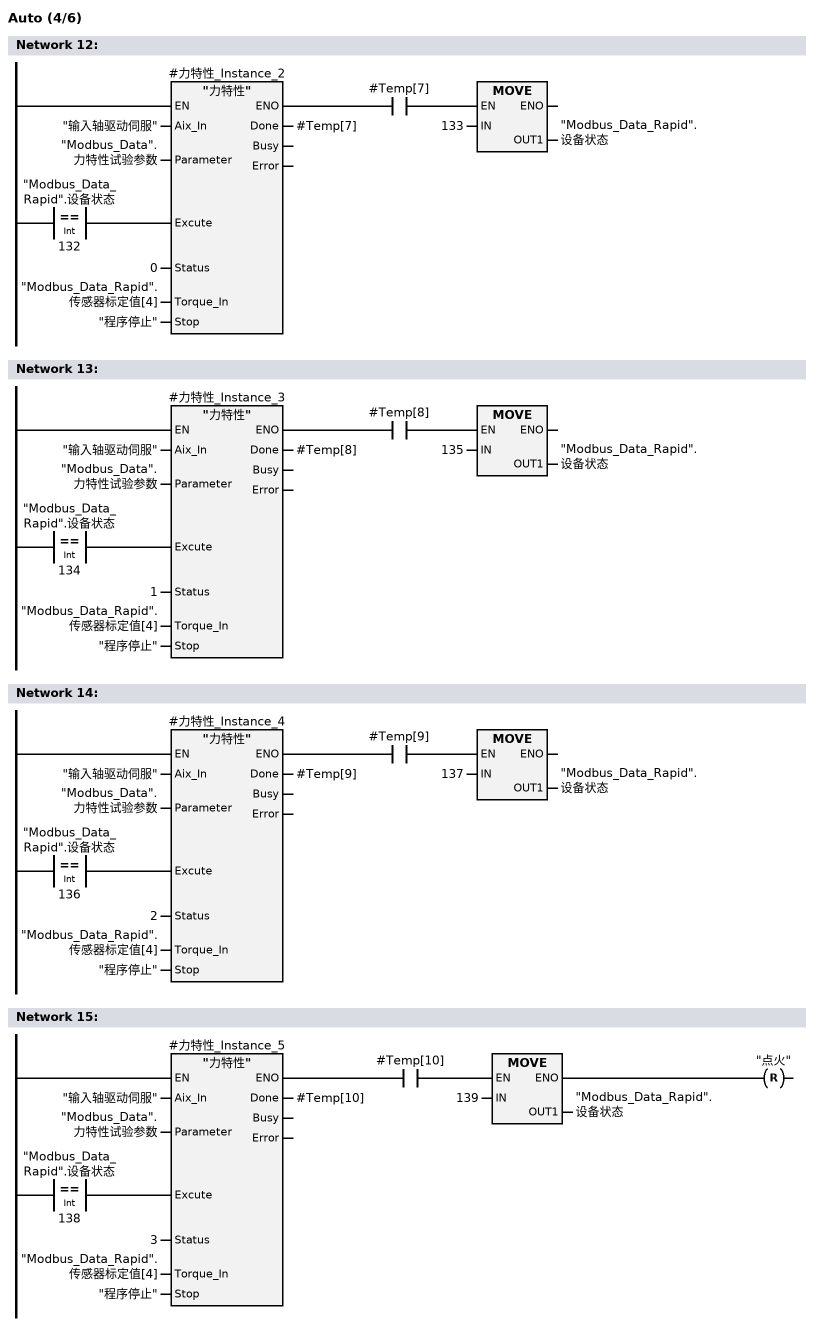
   RUNG wire#powerrail
      #力特性_Instance_2(Excute := wire#w1, Aix_In := "输入轴驱动伺服", Parameter := "Modbus_Data".力特性试验参数, Status := 0, Torque_In := "Modbus_Data_Rapid".传感器标定值[4], Stop := "程序停止", Done => #Temp[7], Busy =>, Error =>)
      Contact( #Temp[7] )
      Move(in := 133, out1 => "Modbus_Data_Rapid".设备状态)
   END_RUNG
   RUNG wire#powerrail
      { S7_Templates := "SrcType := Int" } EQ_Contact(in1 := "Modbus_Data_Rapid".设备状态, in2 := 132)
   END_RUNG wire#w1
   // the same network as SCL:
   #力特性_Instance_2(Aix_In := "输入轴驱动伺服",   // "力特性"
                   Parameter := "Modbus_Data".力特性试验参数,
                   Excute := "Modbus_Data_Rapid".设备状态 = 132,
                   Status := 0,
                   Torque_In := "Modbus_Data_Rapid".传感器标定值[4],
                   Stop := "程序停止",
                   Done => #Temp[7],
                   ENO => #_w1);
   IF #_w1 AND #Temp[7] THEN "Modbus_Data_Rapid".设备状态 := 133; END_IF;
END_REGION

REGION Network 13
   RUNG wire#powerrail
      #力特性_Instance_3(Excute := wire#w1, Aix_In := "输入轴驱动伺服", Parameter := "Modbus_Data".力特性试验参数, Status := 1, Torque_In := "Modbus_Data_Rapid".传感器标定值[4], Stop := "程序停止", Done => #Temp[8], Busy =>, Error =>)
      Contact( #Temp[8] )
      Move(in := 135, out1 => "Modbus_Data_Rapid".设备状态)
   END_RUNG
   RUNG wire#powerrail
      { S7_Templates := "SrcType := Int" } EQ_Contact(in1 := "Modbus_Data_Rapid".设备状态, in2 := 134)
   END_RUNG wire#w1
   // the same network as SCL:
   #力特性_Instance_3(Aix_In := "输入轴驱动伺服",   // "力特性"
                   Parameter := "Modbus_Data".力特性试验参数,
                   Excute := "Modbus_Data_Rapid".设备状态 = 134,
                   Status := 1,
                   Torque_In := "Modbus_Data_Rapid".传感器标定值[4],
                   Stop := "程序停止",
                   Done => #Temp[8],
                   ENO => #_w1);
   IF #_w1 AND #Temp[8] THEN "Modbus_Data_Rapid".设备状态 := 135; END_IF;
END_REGION

REGION Network 14
   RUNG wire#powerrail
      #力特性_Instance_4(Excute := wire#w1, Aix_In := "输入轴驱动伺服", Parameter := "Modbus_Data".力特性试验参数, Status := 2, Torque_In := "Modbus_Data_Rapid".传感器标定值[4], Stop := "程序停止", Done => #Temp[9], Busy =>, Error =>)
      Contact( #Temp[9] )
      Move(in := 137, out1 => "Modbus_Data_Rapid".设备状态)
   END_RUNG
   RUNG wire#powerrail
      { S7_Templates := "SrcType := Int" } EQ_Contact(in1 := "Modbus_Data_Rapid".设备状态, in2 := 136)
   END_RUNG wire#w1
   // the same network as SCL:
   #力特性_Instance_4(Aix_In := "输入轴驱动伺服",   // "力特性"
                   Parameter := "Modbus_Data".力特性试验参数,
                   Excute := "Modbus_Data_Rapid".设备状态 = 136,
                   Status := 2,
                   Torque_In := "Modbus_Data_Rapid".传感器标定值[4],
                   Stop := "程序停止",
                   Done => #Temp[9],
                   ENO => #_w1);
   IF #_w1 AND #Temp[9] THEN "Modbus_Data_Rapid".设备状态 := 137; END_IF;
END_REGION

REGION Network 15
   RUNG wire#powerrail
      #力特性_Instance_5(Excute := wire#w1, Aix_In := "输入轴驱动伺服", Parameter := "Modbus_Data".力特性试验参数, Status := 3, Torque_In := "Modbus_Data_Rapid".传感器标定值[4], Stop := "程序停止", Done => #Temp[10], Busy =>, Error =>)
      Contact( #Temp[10] )
      Move(in := 139, out1 => "Modbus_Data_Rapid".设备状态)
      R_Coil( "点火" )
   END_RUNG
   RUNG wire#powerrail
      { S7_Templates := "SrcType := Int" } EQ_Contact(in1 := "Modbus_Data_Rapid".设备状态, in2 := 138)
   END_RUNG wire#w1
   // the same network as SCL:
   #力特性_Instance_5(Aix_In := "输入轴驱动伺服",   // "力特性"
                   Parameter := "Modbus_Data".力特性试验参数,
                   Excute := "Modbus_Data_Rapid".设备状态 = 138,
                   Status := 3,
                   Torque_In := "Modbus_Data_Rapid".传感器标定值[4],
                   Stop := "程序停止",
                   Done => #Temp[10],
                   ENO => #_w1);
   IF #_w1 AND #Temp[10] THEN
       "Modbus_Data_Rapid".设备状态 := 139;
       "点火" := FALSE;
   END_IF;
END_REGION

REGION Network 16
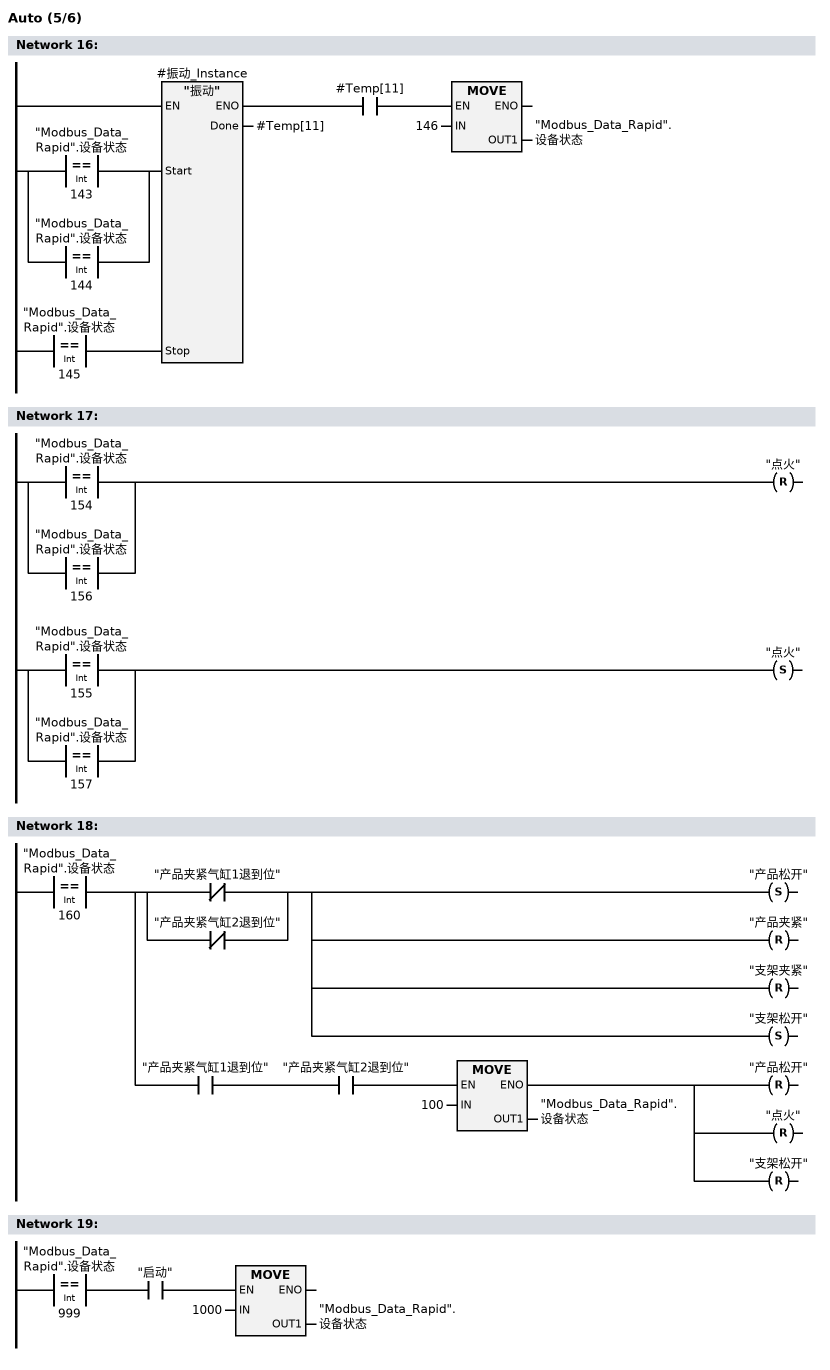
   RUNG wire#powerrail
      #振动_Instance(Start := wire#w1, Stop := wire#w2, Done => #Temp[11])
      Contact( #Temp[11] )
      Move(in := 146, out1 => "Modbus_Data_Rapid".设备状态)
   END_RUNG
   RUNG wire#powerrail
      { S7_Templates := "SrcType := Int" } EQ_Contact(in1 := "Modbus_Data_Rapid".设备状态, in2 := 143)
   END_RUNG wire#w1
   RUNG wire#powerrail
      { S7_Templates := "SrcType := Int" } EQ_Contact(in1 := "Modbus_Data_Rapid".设备状态, in2 := 144)
   END_RUNG wire#w1
   RUNG wire#powerrail
      { S7_Templates := "SrcType := Int" } EQ_Contact(in1 := "Modbus_Data_Rapid".设备状态, in2 := 145)
   END_RUNG wire#w2
   // the same network as SCL:
   #振动_Instance(Start := ("Modbus_Data_Rapid".设备状态 = 143) OR ("Modbus_Data_Rapid".设备状态 = 144),   // "振动"
                Stop := "Modbus_Data_Rapid".设备状态 = 145,
                Done => #Temp[11],
                ENO => #_w1);
   IF #_w1 AND #Temp[11] THEN "Modbus_Data_Rapid".设备状态 := 146; END_IF;
END_REGION

REGION Network 17
   RUNG wire#powerrail
      { S7_Templates := "SrcType := Int" } EQ_Contact(in1 := "Modbus_Data_Rapid".设备状态, in2 := 154)
      wire#w1
      R_Coil( "点火" )
   END_RUNG
   RUNG wire#powerrail
      { S7_Templates := "SrcType := Int" } EQ_Contact(in1 := "Modbus_Data_Rapid".设备状态, in2 := 156)
   END_RUNG wire#w1
   RUNG wire#powerrail
      { S7_Templates := "SrcType := Int" } EQ_Contact(in1 := "Modbus_Data_Rapid".设备状态, in2 := 155)
      wire#w2
      S_Coil( "点火" )
   END_RUNG
   RUNG wire#powerrail
      { S7_Templates := "SrcType := Int" } EQ_Contact(in1 := "Modbus_Data_Rapid".设备状态, in2 := 157)
   END_RUNG wire#w2
   // the same network as SCL:
   IF ("Modbus_Data_Rapid".设备状态 = 154) OR ("Modbus_Data_Rapid".设备状态 = 156) THEN "点火" := FALSE; END_IF;
   IF ("Modbus_Data_Rapid".设备状态 = 155) OR ("Modbus_Data_Rapid".设备状态 = 157) THEN "点火" := TRUE; END_IF;
END_REGION

REGION Network 18
   RUNG wire#powerrail
      { S7_Templates := "SrcType := Int" } EQ_Contact(in1 := "Modbus_Data_Rapid".设备状态, in2 := 160)
      wire#w1
      I_Contact( "产品夹紧气缸1退到位" )
      wire#w2
      S_Coil( "产品松开" )
   END_RUNG
   RUNG wire#w1
      I_Contact( "产品夹紧气缸2退到位" )
   END_RUNG wire#w2
   RUNG wire#w2
      R_Coil( "产品夹紧" )
   END_RUNG
   RUNG wire#w2
      R_Coil( "支架夹紧" )
   END_RUNG
   RUNG wire#w2
      S_Coil( "支架松开" )
   END_RUNG
   RUNG wire#w1
      Contact( "产品夹紧气缸1退到位" )
      Contact( "产品夹紧气缸2退到位" )
      Move(in := 100, out1 => "Modbus_Data_Rapid".设备状态)
      wire#w3
      R_Coil( "产品松开" )
   END_RUNG
   RUNG wire#w3
      R_Coil( "点火" )
   END_RUNG
   RUNG wire#w3
      R_Coil( "支架松开" )
   END_RUNG
   // the same network as SCL:
   #_w1 := "Modbus_Data_Rapid".设备状态 = 160;
   IF #_w1 AND (NOT "产品夹紧气缸1退到位" OR NOT "产品夹紧气缸2退到位") THEN
       "产品松开" := TRUE;
       "产品夹紧" := FALSE;
       "支架夹紧" := FALSE;
       "支架松开" := TRUE;
   END_IF;
   IF #_w1 AND "产品夹紧气缸1退到位" AND "产品夹紧气缸2退到位" THEN
       "Modbus_Data_Rapid".设备状态 := 100;
       "产品松开" := FALSE;
       "点火" := FALSE;
       "支架松开" := FALSE;
   END_IF;
END_REGION

REGION Network 19
   RUNG wire#powerrail
      { S7_Templates := "SrcType := Int" } EQ_Contact(in1 := "Modbus_Data_Rapid".设备状态, in2 := 999)
      Contact( "启动" )
      Move(in := 1000, out1 => "Modbus_Data_Rapid".设备状态)
   END_RUNG
   // the same network as SCL:
   IF ("Modbus_Data_Rapid".设备状态 = 999) AND "启动" THEN "Modbus_Data_Rapid".设备状态 := 1000; END_IF;
END_REGION

REGION Network 20
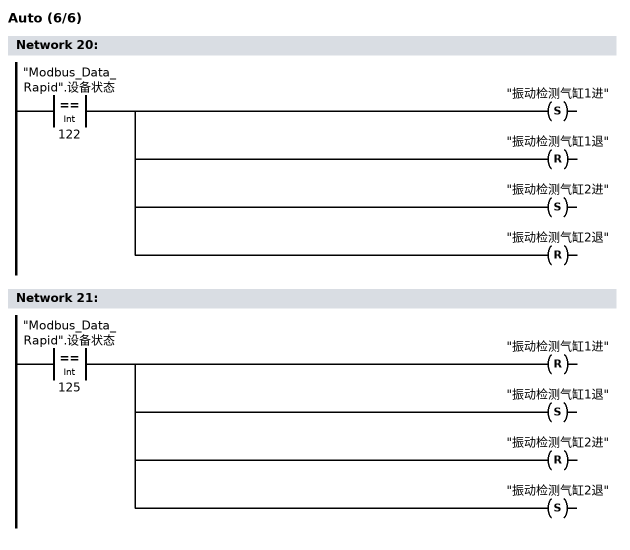
   RUNG wire#powerrail
      { S7_Templates := "SrcType := Int" } EQ_Contact(in1 := "Modbus_Data_Rapid".设备状态, in2 := 122)
      wire#w1
      S_Coil( "振动检测气缸1进" )
   END_RUNG
   RUNG wire#w1
      R_Coil( "振动检测气缸1退" )
   END_RUNG
   RUNG wire#w1
      S_Coil( "振动检测气缸2进" )
   END_RUNG
   RUNG wire#w1
      R_Coil( "振动检测气缸2退" )
   END_RUNG
   // the same network as SCL:
   IF "Modbus_Data_Rapid".设备状态 = 122 THEN
       "振动检测气缸1进" := TRUE;
       "振动检测气缸1退" := FALSE;
       "振动检测气缸2进" := TRUE;
       "振动检测气缸2退" := FALSE;
   END_IF;
END_REGION

REGION Network 21
   RUNG wire#powerrail
      { S7_Templates := "SrcType := Int" } EQ_Contact(in1 := "Modbus_Data_Rapid".设备状态, in2 := 125)
      wire#w1
      R_Coil( "振动检测气缸1进" )
   END_RUNG
   RUNG wire#w1
      S_Coil( "振动检测气缸1退" )
   END_RUNG
   RUNG wire#w1
      R_Coil( "振动检测气缸2进" )
   END_RUNG
   RUNG wire#w1
      S_Coil( "振动检测气缸2退" )
   END_RUNG
   // the same network as SCL:
   IF "Modbus_Data_Rapid".设备状态 = 125 THEN
       "振动检测气缸1进" := FALSE;
       "振动检测气缸1退" := TRUE;
       "振动检测气缸2进" := FALSE;
       "振动检测气缸2退" := TRUE;
   END_IF;
END_REGION
END_FUNCTION_BLOCK

FUNCTION_BLOCK "力特性"   // FB11, LAD
{ S7_Optimized_Access := 'TRUE' }
VERSION : 0.1
   VAR_INPUT
      Aix_In : TO_PositioningAxis;
      Parameter : "Test_Input&Output_Characteristics_CFG";
      Excute : Bool;
      Status : Byte;
      Torque_In : Real;
      Stop : Bool;
   END_VAR
   VAR_OUTPUT
      Done : Bool;
      Busy : Bool;
      Error : Bool;
   END_VAR
   VAR
      "Step" : Int;
      Switch_Torque : Real;
      Test_Velocity : Real;
      Temp : Array[0..7] of Bool;
      MC_Halt_Instance : MC_Halt;
      MC_Home_Instance : MC_Home;
      MC_MoveVelocity_Instance : MC_MoveVelocity;
   END_VAR
   VAR_TEMP   // added for the SCL form of the ladder/FBD networks
      _w1 : Bool;
   END_VAR
BEGIN

REGION Network 1
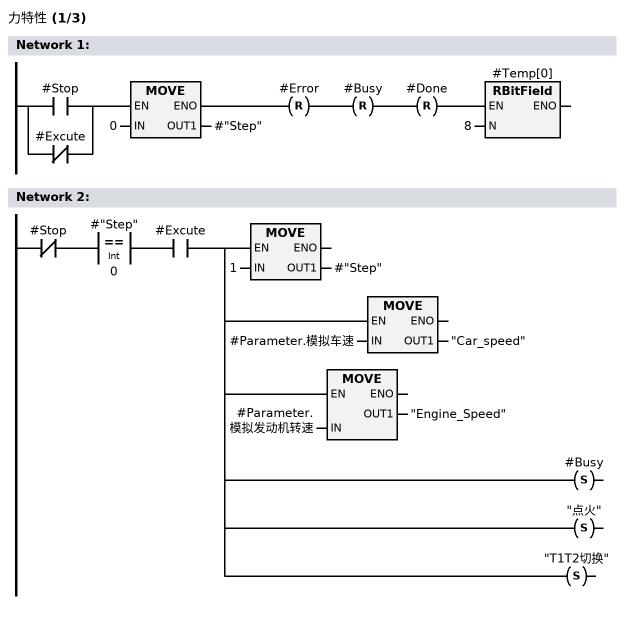
   // no SCL statement known for RBitField: written as a call
   IF #Stop OR NOT #Excute THEN
       #"Step" := 0;
       #Error := FALSE;
       #Busy := FALSE;
       #Done := FALSE;
       RBitField(n := 8, operand := #Temp[0]);
   END_IF;
END_REGION

REGION Network 2
   RUNG wire#powerrail
      I_Contact( #Stop )
      { S7_Templates := "SrcType := Int" } EQ_Contact(in1 := #"Step", in2 := 0)
      Contact( #Excute )
      wire#w1
      Move(in := 1, out1 => #"Step")
   END_RUNG
   RUNG wire#w1
      Move(in := #Parameter.模拟车速, out1 => "Car_speed")
   END_RUNG
   RUNG wire#w1
      Move(in := #Parameter.模拟发动机转速, out1 => "Engine_Speed")
   END_RUNG
   RUNG wire#w1
      S_Coil( #Busy )
   END_RUNG
   RUNG wire#w1
      S_Coil( "点火" )
   END_RUNG
   RUNG wire#w1
      S_Coil( "T1T2切换" )
   END_RUNG
   // the same network as SCL:
   #_w1 := NOT #Stop AND (#"Step" = 0) AND #Excute;
   IF #_w1 THEN
       #"Step" := 1;
       "Car_speed" := #Parameter.模拟车速;
       "Engine_Speed" := #Parameter.模拟发动机转速;
       #Busy := TRUE;
       "点火" := TRUE;
       "T1T2切换" := TRUE;
   END_IF;
END_REGION

REGION Network 3
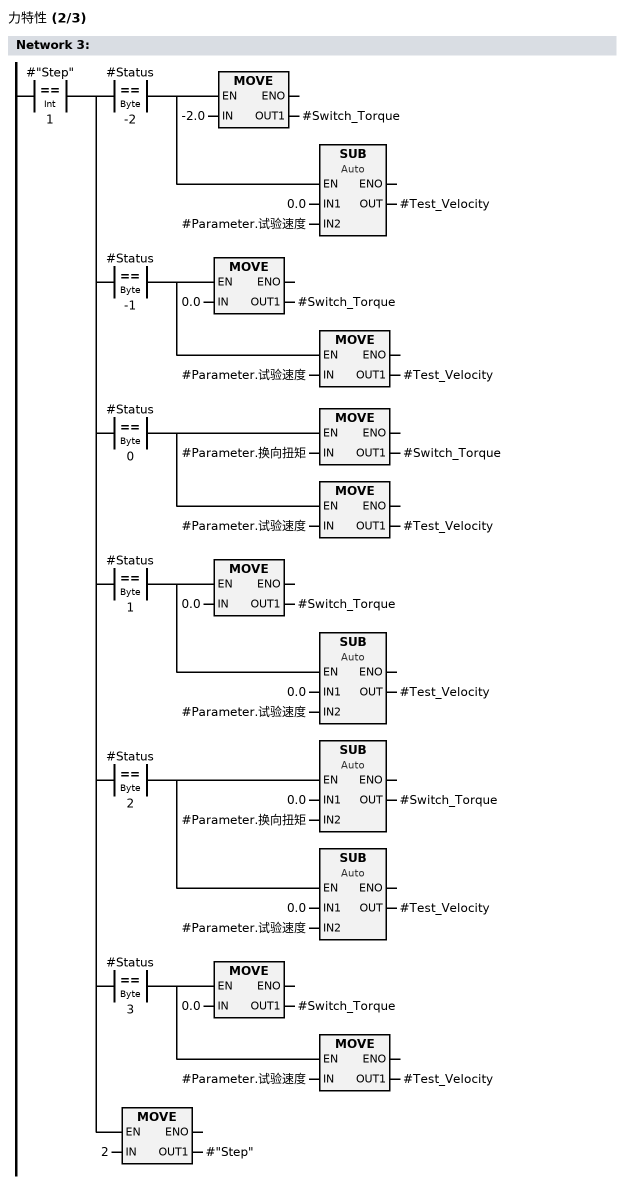
   RUNG wire#powerrail
      { S7_Templates := "SrcType := Int" } EQ_Contact(in1 := #"Step", in2 := 1)
      wire#w1
      { S7_Templates := "SrcType := Byte" } EQ_Contact(in1 := #Status, in2 := -2)
      wire#w2
      Move(in := -2.0, out1 => #Switch_Torque)
   END_RUNG
   RUNG wire#w2
      Sub(in1 := 0.0, in2 := #Parameter.试验速度, out => #Test_Velocity)
   END_RUNG
   RUNG wire#w1
      { S7_Templates := "SrcType := Byte" } EQ_Contact(in1 := #Status, in2 := -1)
      wire#w3
      Move(in := 0.0, out1 => #Switch_Torque)
   END_RUNG
   RUNG wire#w3
      Move(in := #Parameter.试验速度, out1 => #Test_Velocity)
   END_RUNG
   RUNG wire#w1
      { S7_Templates := "SrcType := Byte" } EQ_Contact(in1 := #Status, in2 := 0)
      wire#w4
      Move(in := #Parameter.换向扭矩, out1 => #Switch_Torque)
   END_RUNG
   RUNG wire#w4
      Move(in := #Parameter.试验速度, out1 => #Test_Velocity)
   END_RUNG
   RUNG wire#w1
      { S7_Templates := "SrcType := Byte" } EQ_Contact(in1 := #Status, in2 := 1)
      wire#w5
      Move(in := 0.0, out1 => #Switch_Torque)
   END_RUNG
   RUNG wire#w5
      Sub(in1 := 0.0, in2 := #Parameter.试验速度, out => #Test_Velocity)
   END_RUNG
   RUNG wire#w1
      { S7_Templates := "SrcType := Byte" } EQ_Contact(in1 := #Status, in2 := 2)
      wire#w6
      Sub(in1 := 0.0, in2 := #Parameter.换向扭矩, out => #Switch_Torque)
   END_RUNG
   RUNG wire#w6
      Sub(in1 := 0.0, in2 := #Parameter.试验速度, out => #Test_Velocity)
   END_RUNG
   RUNG wire#w1
      { S7_Templates := "SrcType := Byte" } EQ_Contact(in1 := #Status, in2 := 3)
      wire#w7
      Move(in := 0.0, out1 => #Switch_Torque)
   END_RUNG
   RUNG wire#w7
      Move(in := #Parameter.试验速度, out1 => #Test_Velocity)
   END_RUNG
   RUNG wire#w1
      Move(in := 2, out1 => #"Step")
   END_RUNG
   // the same network as SCL:
   #_w1 := #"Step" = 1;
   IF #_w1 AND (#Status = (-2)) THEN
       #Switch_Torque := -2.0;
       #Test_Velocity := 0.0 - #Parameter.试验速度;
   END_IF;
   IF #_w1 AND (#Status = (-1)) THEN
       #Switch_Torque := 0.0;
       #Test_Velocity := #Parameter.试验速度;
   END_IF;
   IF #_w1 AND (#Status = 0) THEN
       #Switch_Torque := #Parameter.换向扭矩;
       #Test_Velocity := #Parameter.试验速度;
   END_IF;
   IF #_w1 AND (#Status = 1) THEN
       #Switch_Torque := 0.0;
       #Test_Velocity := 0.0 - #Parameter.试验速度;
   END_IF;
   IF #_w1 AND (#Status = 2) THEN
       #Switch_Torque := 0.0 - #Parameter.换向扭矩;
       #Test_Velocity := 0.0 - #Parameter.试验速度;
   END_IF;
   IF #_w1 AND (#Status = 3) THEN
       #Switch_Torque := 0.0;
       #Test_Velocity := #Parameter.试验速度;
   END_IF;
   IF #_w1 THEN #"Step" := 2; END_IF;
END_REGION

REGION Network 4
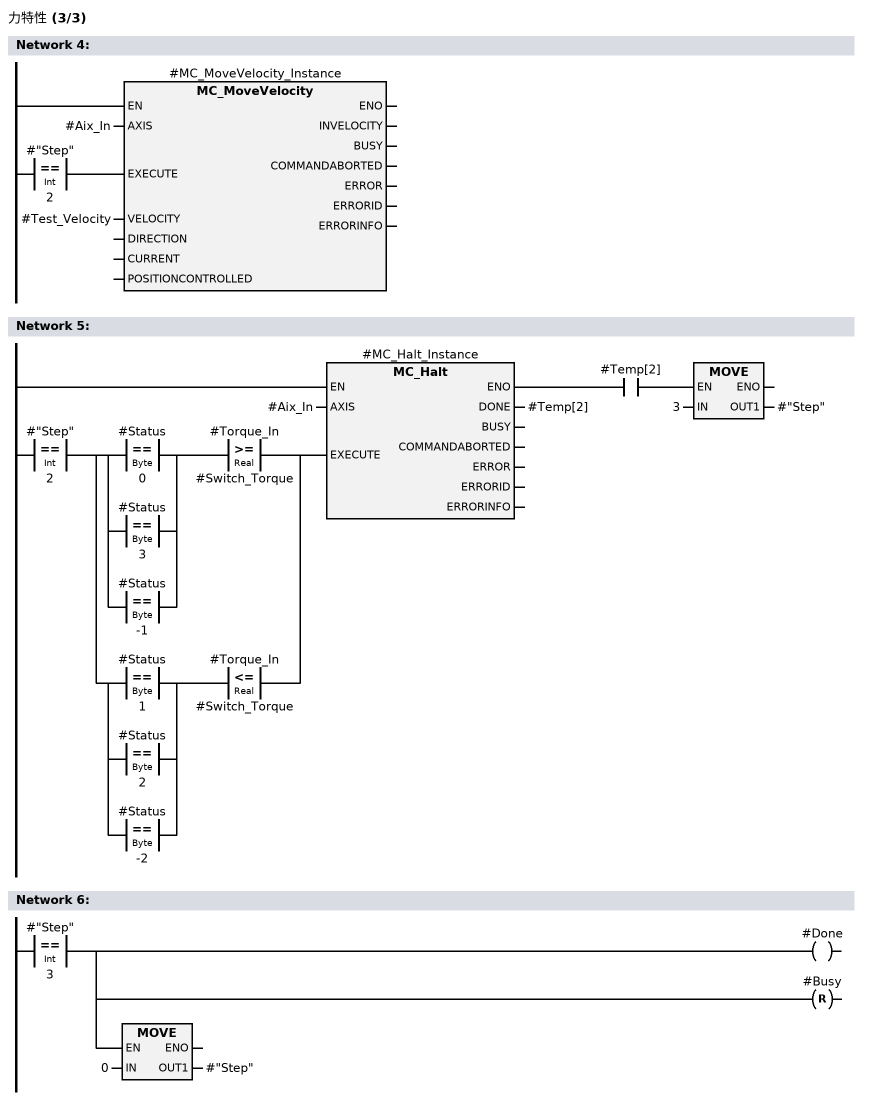
   #MC_MoveVelocity_Instance(Axis := #Aix_In, Execute := #"Step" = 2, Velocity := #Test_Velocity);   // MC_MoveVelocity
END_REGION

REGION Network 5
   // ENO of a box is taken as its EN; it also drops when the box reports an error
   #MC_Halt_Instance(Axis := #Aix_In,   // MC_Halt
                     Execute := (#"Step" = 2) AND ((((#Status = 0) OR (#Status = 3) OR (#Status = (-1))) AND (#Torque_In >= #Switch_Torque)) OR (((#Status = 1) OR (#Status = 2) OR (#Status = (-2))) AND (#Torque_In <= #Switch_Torque))),
                     Done => #Temp[2]);
   IF #Temp[2] THEN #"Step" := 3; END_IF;
END_REGION

REGION Network 6
   RUNG wire#powerrail
      { S7_Templates := "SrcType := Int" } EQ_Contact(in1 := #"Step", in2 := 3)
      wire#w1
      Coil( #Done )
   END_RUNG
   RUNG wire#w1
      R_Coil( #Busy )
   END_RUNG
   RUNG wire#w1
      Move(in := 0, out1 => #"Step")
   END_RUNG
   // the same network as SCL:
   #Done := #"Step" = 3;
   IF #Done THEN
       #Busy := FALSE;
       #"Step" := 0;
   END_IF;
END_REGION
END_FUNCTION_BLOCK

FUNCTION_BLOCK "振动"   // FB12, LAD
{ S7_Optimized_Access := 'TRUE' }
VERSION : 0.1
   VAR_INPUT
      Start : Bool;
      Stop : Bool;
   END_VAR
   VAR_OUTPUT
      Done : Bool;
   END_VAR
   VAR
      "Step" : Int;
      IEC_Timer_0_Instance : TON_TIME;
   END_VAR
BEGIN

REGION Network 1
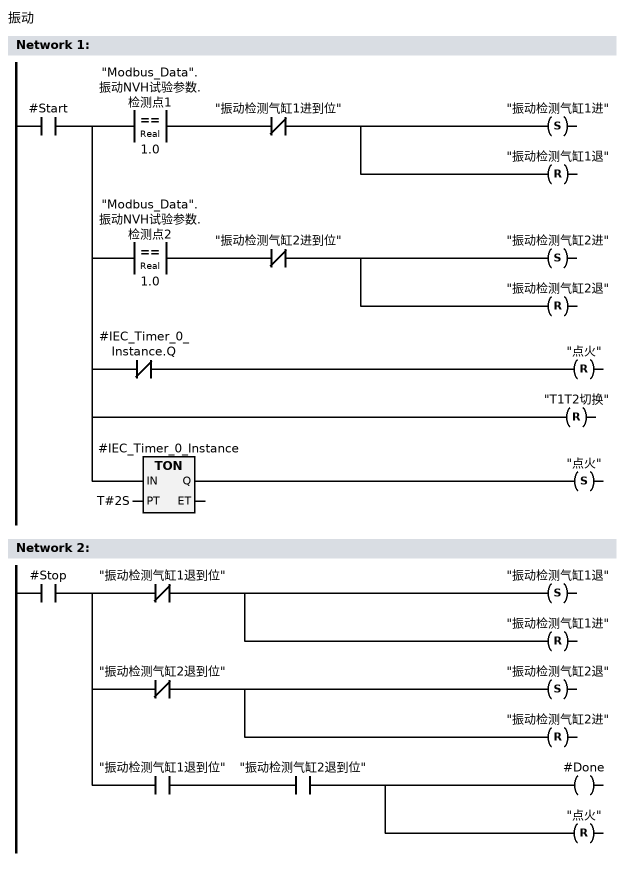
   IF #Start AND ("Modbus_Data".振动NVH试验参数.检测点1 = 1.0) AND NOT "振动检测气缸1进到位" THEN
       "振动检测气缸1进" := TRUE;
       "振动检测气缸1退" := FALSE;
   END_IF;
   IF #Start AND ("Modbus_Data".振动NVH试验参数.检测点2 = 1.0) AND NOT "振动检测气缸2进到位" THEN
       "振动检测气缸2进" := TRUE;
       "振动检测气缸2退" := FALSE;
   END_IF;
   IF #Start AND NOT #IEC_Timer_0_Instance.Q THEN "点火" := FALSE; END_IF;
   IF #Start THEN "T1T2切换" := FALSE; END_IF;
   #IEC_Timer_0_Instance(IN := #Start, PT := T#2S);   // TON
   IF #IEC_Timer_0_Instance.Q THEN "点火" := TRUE; END_IF;
END_REGION

REGION Network 2
   RUNG wire#powerrail
      Contact( #Stop )
      wire#w1
      I_Contact( "振动检测气缸1退到位" )
      wire#w2
      S_Coil( "振动检测气缸1退" )
   END_RUNG
   RUNG wire#w2
      R_Coil( "振动检测气缸1进" )
   END_RUNG
   RUNG wire#w1
      I_Contact( "振动检测气缸2退到位" )
      wire#w3
      S_Coil( "振动检测气缸2退" )
   END_RUNG
   RUNG wire#w3
      R_Coil( "振动检测气缸2进" )
   END_RUNG
   RUNG wire#w1
      Contact( "振动检测气缸1退到位" )
      Contact( "振动检测气缸2退到位" )
      wire#w4
      Coil( #Done )
   END_RUNG
   RUNG wire#w4
      R_Coil( "点火" )
   END_RUNG
   // the same network as SCL:
   IF #Stop AND NOT "振动检测气缸1退到位" THEN
       "振动检测气缸1退" := TRUE;
       "振动检测气缸1进" := FALSE;
   END_IF;
   IF #Stop AND NOT "振动检测气缸2退到位" THEN
       "振动检测气缸2退" := TRUE;
       "振动检测气缸2进" := FALSE;
   END_IF;
   #Done := #Stop AND "振动检测气缸1退到位" AND "振动检测气缸2退到位";
   IF #Done THEN "点火" := FALSE; END_IF;
END_REGION
END_FUNCTION_BLOCK

FUNCTION "Analog To Project amount" : Void   // FC1, LAD
{ S7_Optimized_Access := 'TRUE' }
VERSION : 0.1
   VAR_INPUT
      Analog : Int;
      Min_Value : Real;
      Max_Value : Real;
   END_VAR
   VAR_OUTPUT
      Project_amount : Real;
   END_VAR
   VAR_TEMP
      Temp_Value : Real;
   END_VAR
BEGIN

REGION Network 1
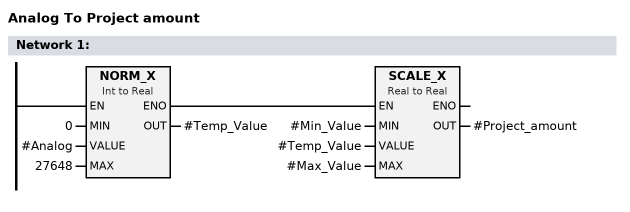
   RUNG wire#powerrail
      { S7_Templates := "[SrcType := Int, DestType := Real]" } Normalize(min := 0, value := #Analog, max := 27648, out => #Temp_Value)
      { S7_Templates := "[SrcType := Real, DestType := Real]" } Scale(min := #Min_Value, value := #Temp_Value, max := #Max_Value, out => #Project_amount)
   END_RUNG
   // the same network as SCL:
   #Temp_Value := NORM_X(MIN := 0, VALUE := #Analog, MAX := 27648);
   #Project_amount := SCALE_X(MIN := #Min_Value, VALUE := #Temp_Value, MAX := #Max_Value);
END_REGION
END_FUNCTION

FUNCTION "encoder" : Void   // FC2, LAD
{ S7_Optimized_Access := 'TRUE' }
VERSION : 0.1
   VAR_INPUT
      encoder : DInt;
   END_VAR
   VAR_OUTPUT
      angle : Real;
   END_VAR
   VAR_TEMP
      Temp_Value : DInt;
      Temp_Value2 : DInt;
   END_VAR
BEGIN

REGION Network 1
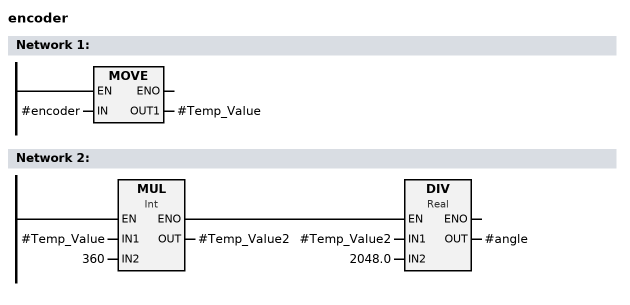
   RUNG wire#powerrail
      Move(in := #encoder, out1 => #Temp_Value)
   END_RUNG
   // the same network as SCL:
   #Temp_Value := #encoder;
END_REGION

REGION Network 2
   RUNG wire#powerrail
      { S7_Templates := "SrcType := Int" } Mul(in1 := #Temp_Value, in2 := 360, out => #Temp_Value2)
      { S7_Templates := "SrcType := Real" } Div(in1 := #Temp_Value2, in2 := 2048.0, out => #angle)
   END_RUNG
   // the same network as SCL:
   #Temp_Value2 := #Temp_Value * 360;
   #angle := #Temp_Value2 / 2048.0;
END_REGION
END_FUNCTION

FUNCTION "Project amount To Analog" : Void   // FC3, LAD
{ S7_Optimized_Access := 'TRUE' }
VERSION : 0.1
   VAR_INPUT
      Project_amount : Real;
      Project_amount_min : Real;
      Project_amount_max : Real;
      Analog_min : Int;
      Analog_max : Int;
   END_VAR
   VAR_OUTPUT
      Analog : Int;
   END_VAR
   VAR_TEMP
      temp_out : Real;
   END_VAR
BEGIN

REGION Network 1
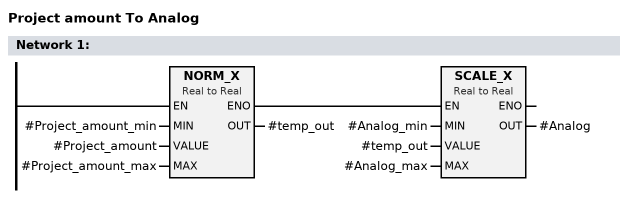
   RUNG wire#powerrail
      { S7_Templates := "[SrcType := Real, DestType := Real]" } Normalize(min := #Project_amount_min, value := #Project_amount, max := #Project_amount_max, out => #temp_out)
      { S7_Templates := "[SrcType := Real, DestType := Real]" } Scale(min := #Analog_min, value := #temp_out, max := #Analog_max, out => #Analog)
   END_RUNG
   // the same network as SCL:
   #temp_out := NORM_X(MIN := #Project_amount_min, VALUE := #Project_amount, MAX := #Project_amount_max);
   #Analog := SCALE_X(MIN := #Analog_min, VALUE := #temp_out, MAX := #Analog_max);
END_REGION
END_FUNCTION

ORGANIZATION_BLOCK "Main"   // OB1, LAD, ProgramCycle
TITLE = "Main Program Sweep (Cycle)"
{ S7_Optimized_Access := 'TRUE' }
VERSION : 0.1
   VAR_INPUT
      Initial_Call : Bool;   // Initial call of this OB
      Remanence : Bool;   // =True, if remanent data are available
   END_VAR
   VAR_TEMP
      电压 : Real;
   END_VAR
   VAR_TEMP   // added for the SCL form of the ladder/FBD networks
      _w1 : Bool;
   END_VAR
BEGIN

REGION Network 1
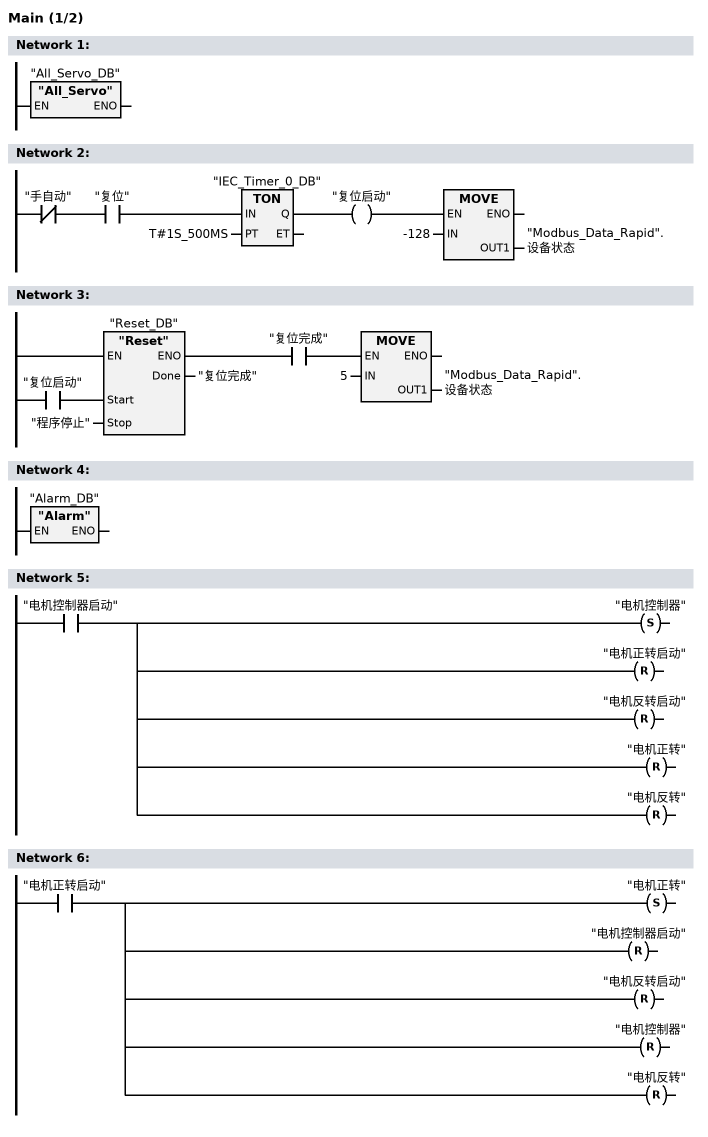
   RUNG wire#powerrail
      "All_Servo_DB"()
   END_RUNG
   // the same network as SCL:
   "All_Servo_DB"();   // "All_Servo"
END_REGION

REGION Network 2
   "IEC_Timer_0_DB".TON(IN := NOT "手自动" AND "复位", PT := T#1S_500MS);
   "复位启动" := "IEC_Timer_0_DB".Q;
   IF "IEC_Timer_0_DB".Q THEN "Modbus_Data_Rapid".设备状态 := -128; END_IF;
END_REGION

REGION Network 3
   RUNG wire#powerrail
      "Reset_DB"(Start := wire#w1, Stop := "程序停止", Done => "复位完成")
      Contact( "复位完成" )
      Move(in := 5, out1 => "Modbus_Data_Rapid".设备状态)
   END_RUNG
   RUNG wire#powerrail
      Contact( "复位启动" )
   END_RUNG wire#w1
   // the same network as SCL:
   "Reset_DB"(Start := "复位启动", Stop := "程序停止", Done => "复位完成", ENO => #_w1);   // "Reset"
   IF #_w1 AND "复位完成" THEN "Modbus_Data_Rapid".设备状态 := 5; END_IF;
END_REGION

REGION Network 4
   RUNG wire#powerrail
      "Alarm_DB"()
   END_RUNG
   // the same network as SCL:
   "Alarm_DB"();   // "Alarm"
END_REGION

REGION Network 5
   RUNG wire#powerrail
      Contact( "电机控制器启动" )
      wire#w1
      S_Coil( "电机控制器" )
   END_RUNG
   RUNG wire#w1
      R_Coil( "电机正转启动" )
   END_RUNG
   RUNG wire#w1
      R_Coil( "电机反转启动" )
   END_RUNG
   RUNG wire#w1
      R_Coil( "电机正转" )
   END_RUNG
   RUNG wire#w1
      R_Coil( "电机反转" )
   END_RUNG
   // the same network as SCL:
   IF "电机控制器启动" THEN
       "电机控制器" := TRUE;
       "电机正转启动" := FALSE;
       "电机反转启动" := FALSE;
       "电机正转" := FALSE;
       "电机反转" := FALSE;
   END_IF;
END_REGION

REGION Network 6
   RUNG wire#powerrail
      Contact( "电机正转启动" )
      wire#w1
      S_Coil( "电机正转" )
   END_RUNG
   RUNG wire#w1
      R_Coil( "电机控制器启动" )
   END_RUNG
   RUNG wire#w1
      R_Coil( "电机反转启动" )
   END_RUNG
   RUNG wire#w1
      R_Coil( "电机控制器" )
   END_RUNG
   RUNG wire#w1
      R_Coil( "电机反转" )
   END_RUNG
   // the same network as SCL:
   IF "电机正转启动" THEN
       "电机正转" := TRUE;
       "电机控制器启动" := FALSE;
       "电机反转启动" := FALSE;
       "电机控制器" := FALSE;
       "电机反转" := FALSE;
   END_IF;
END_REGION

REGION Network 7
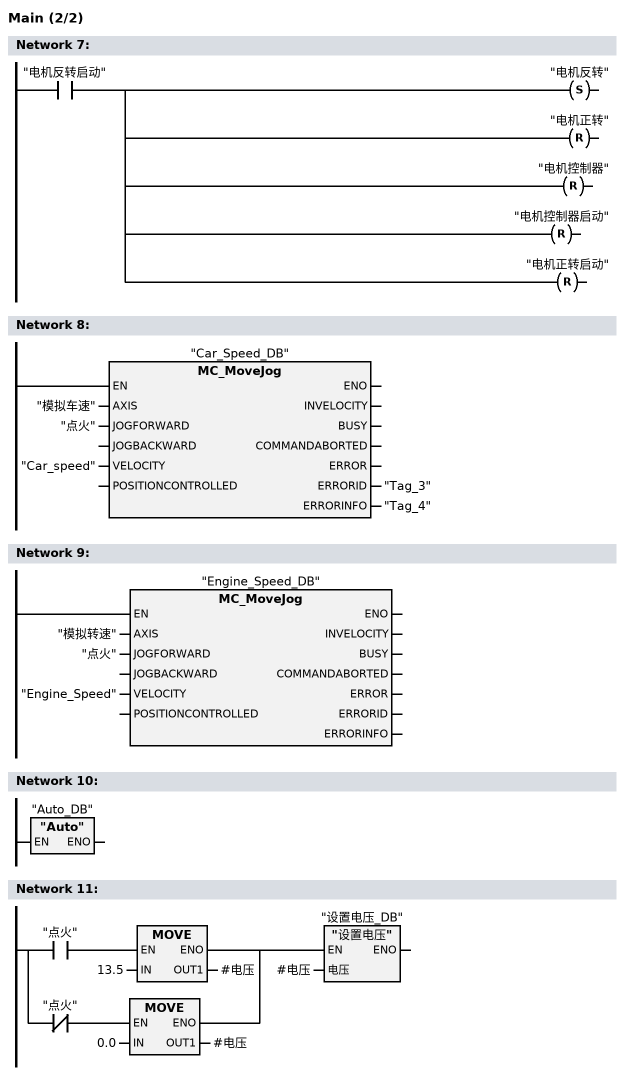
   RUNG wire#powerrail
      Contact( "电机反转启动" )
      wire#w1
      S_Coil( "电机反转" )
   END_RUNG
   RUNG wire#w1
      R_Coil( "电机正转" )
   END_RUNG
   RUNG wire#w1
      R_Coil( "电机控制器" )
   END_RUNG
   RUNG wire#w1
      R_Coil( "电机控制器启动" )
   END_RUNG
   RUNG wire#w1
      R_Coil( "电机正转启动" )
   END_RUNG
   // the same network as SCL:
   IF "电机反转启动" THEN
       "电机反转" := TRUE;
       "电机正转" := FALSE;
       "电机控制器" := FALSE;
       "电机控制器启动" := FALSE;
       "电机正转启动" := FALSE;
   END_IF;
END_REGION

REGION Network 8
   "Car_Speed_DB"(Axis := "模拟车速",   // MC_MoveJog
                  JogForward := "点火",
                  Velocity := "Car_speed",
                  ErrorID => "Tag_3",
                  ErrorInfo => "Tag_4");
END_REGION

REGION Network 9
   "Engine_Speed_DB"(Axis := "模拟转速", JogForward := "点火", Velocity := "Engine_Speed");   // MC_MoveJog
END_REGION

REGION Network 10
   RUNG wire#powerrail
      "Auto_DB"()
   END_RUNG
   // the same network as SCL:
   "Auto_DB"();   // "Auto"
END_REGION

REGION Network 11
   RUNG wire#powerrail
      Contact( "点火" )
      Move(in := 13.5, out1 => #电压)
      wire#w1
      "设置电压_DB"(电压 := #电压)
   END_RUNG
   RUNG wire#powerrail
      I_Contact( "点火" )
      Move(in := 0.0, out1 => #电压)
   END_RUNG wire#w1
   // the same network as SCL:
   IF "点火" THEN #电压 := 13.5; END_IF;
   IF NOT "点火" THEN #电压 := 0.0; END_IF;
   IF "点火" OR NOT "点火" THEN
       "设置电压_DB"(电压 := #电压);   // "设置电压"
   END_IF;
END_REGION
END_ORGANIZATION_BLOCK

ORGANIZATION_BLOCK "Cyclic interrupt_10ms"   // OB30, LAD, CyclicInterrupt
{ S7_Optimized_Access := 'TRUE' }
VERSION : 0.1
   VAR_INPUT
      Initial_Call : Bool;   // Initial call of this OB
      Event_Count : Int;   // Events discarded
   END_VAR
   VAR_TEMP   // added for the SCL form of the ladder/FBD networks
      _w1 : Bool;
   END_VAR
BEGIN

REGION Network 1
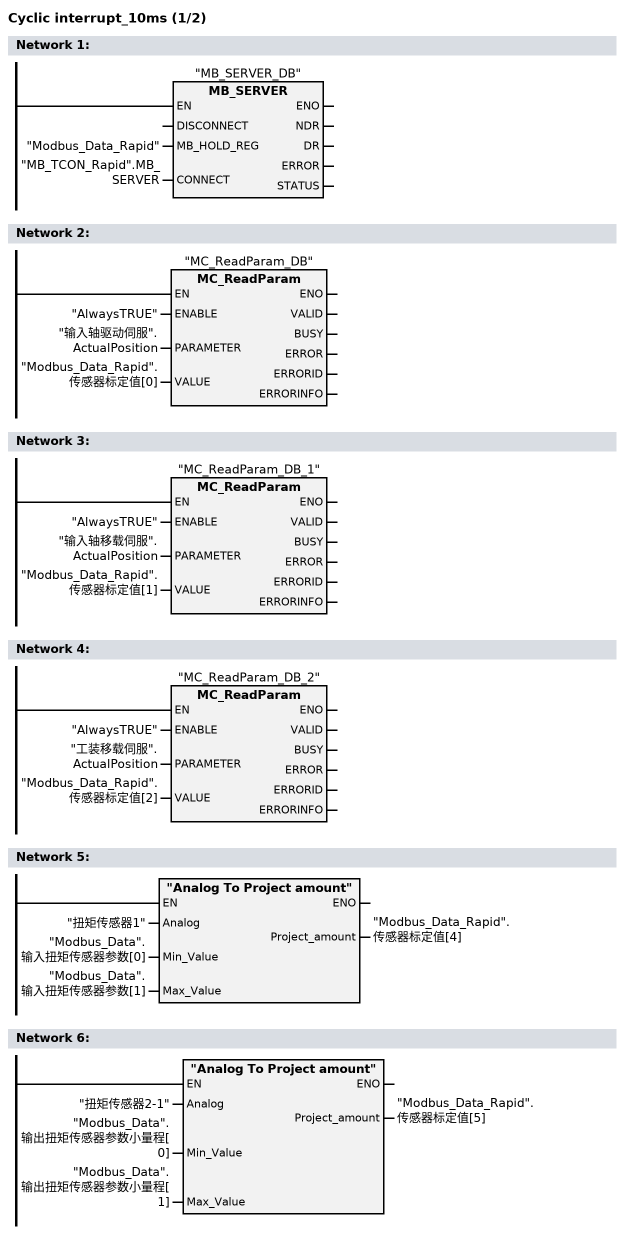
   "MB_SERVER_DB"(MB_HOLD_REG := "Modbus_Data_Rapid", CONNECT := "MB_TCON_Rapid".MB_SERVER);   // MB_SERVER
END_REGION

REGION Network 2
   "MC_ReadParam_DB"(Enable := "AlwaysTRUE",   // MC_ReadParam
                     Parameter := "输入轴驱动伺服".ActualPosition,
                     Value := "Modbus_Data_Rapid".传感器标定值[0]);
END_REGION

REGION Network 3
   "MC_ReadParam_DB_1"(Enable := "AlwaysTRUE",   // MC_ReadParam
                       Parameter := "输入轴移载伺服".ActualPosition,
                       Value := "Modbus_Data_Rapid".传感器标定值[1]);
END_REGION

REGION Network 4
   "MC_ReadParam_DB_2"(Enable := "AlwaysTRUE",   // MC_ReadParam
                       Parameter := "工装移载伺服".ActualPosition,
                       Value := "Modbus_Data_Rapid".传感器标定值[2]);
END_REGION

REGION Network 5
   RUNG wire#powerrail
      "Analog To Project amount"(Analog := "扭矩传感器1", Min_Value := "Modbus_Data".输入扭矩传感器参数[0], Max_Value := "Modbus_Data".输入扭矩传感器参数[1], Project_amount => "Modbus_Data_Rapid".传感器标定值[4])
   END_RUNG
   // the same network as SCL:
   "Analog To Project amount"(Analog := "扭矩传感器1",
                           Min_Value := "Modbus_Data".输入扭矩传感器参数[0],
                           Max_Value := "Modbus_Data".输入扭矩传感器参数[1],
                           Project_amount => "Modbus_Data_Rapid".传感器标定值[4]);
END_REGION

REGION Network 6
   RUNG wire#powerrail
      "Analog To Project amount"(Analog := "扭矩传感器2-1", Min_Value := "Modbus_Data".输出扭矩传感器参数小量程[0], Max_Value := "Modbus_Data".输出扭矩传感器参数小量程[1], Project_amount => "Modbus_Data_Rapid".传感器标定值[5])
   END_RUNG
   // the same network as SCL:
   "Analog To Project amount"(Analog := "扭矩传感器2-1",
                           Min_Value := "Modbus_Data".输出扭矩传感器参数小量程[0],
                           Max_Value := "Modbus_Data".输出扭矩传感器参数小量程[1],
                           Project_amount => "Modbus_Data_Rapid".传感器标定值[5]);
END_REGION

REGION Network 7
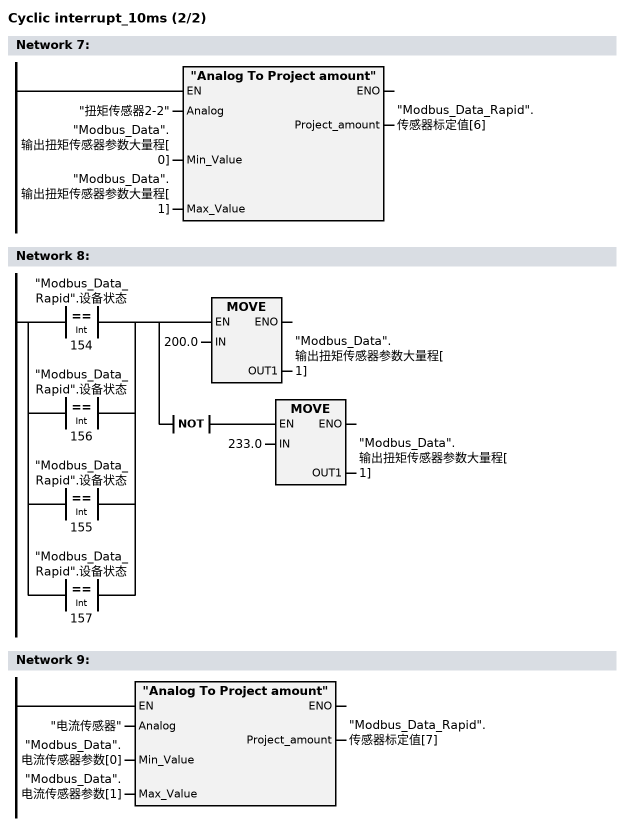
   RUNG wire#powerrail
      "Analog To Project amount"(Analog := "扭矩传感器2-2", Min_Value := "Modbus_Data".输出扭矩传感器参数大量程[0], Max_Value := "Modbus_Data".输出扭矩传感器参数大量程[1], Project_amount => "Modbus_Data_Rapid".传感器标定值[6])
   END_RUNG
   // the same network as SCL:
   "Analog To Project amount"(Analog := "扭矩传感器2-2",
                           Min_Value := "Modbus_Data".输出扭矩传感器参数大量程[0],
                           Max_Value := "Modbus_Data".输出扭矩传感器参数大量程[1],
                           Project_amount => "Modbus_Data_Rapid".传感器标定值[6]);
END_REGION

REGION Network 8
   RUNG wire#powerrail
      { S7_Templates := "SrcType := Int" } EQ_Contact(in1 := "Modbus_Data_Rapid".设备状态, in2 := 154)
      wire#w1
      Move(in := 200.0, out1 => "Modbus_Data".输出扭矩传感器参数大量程[1])
   END_RUNG
   RUNG wire#powerrail
      { S7_Templates := "SrcType := Int" } EQ_Contact(in1 := "Modbus_Data_Rapid".设备状态, in2 := 156)
   END_RUNG wire#w1
   RUNG wire#powerrail
      { S7_Templates := "SrcType := Int" } EQ_Contact(in1 := "Modbus_Data_Rapid".设备状态, in2 := 155)
   END_RUNG wire#w1
   RUNG wire#powerrail
      { S7_Templates := "SrcType := Int" } EQ_Contact(in1 := "Modbus_Data_Rapid".设备状态, in2 := 157)
   END_RUNG wire#w1
   RUNG wire#w1
      Not()
      Move(in := 233.0, out1 => "Modbus_Data".输出扭矩传感器参数大量程[1])
   END_RUNG
   // the same network as SCL:
   #_w1 := ("Modbus_Data_Rapid".设备状态 = 154) OR ("Modbus_Data_Rapid".设备状态 = 156) OR ("Modbus_Data_Rapid".设备状态 = 155) OR ("Modbus_Data_Rapid".设备状态 = 157);
   IF #_w1 THEN "Modbus_Data".输出扭矩传感器参数大量程[1] := 200.0; END_IF;
   IF NOT #_w1 THEN "Modbus_Data".输出扭矩传感器参数大量程[1] := 233.0; END_IF;
END_REGION

REGION Network 9
   RUNG wire#powerrail
      "Analog To Project amount"(Analog := "电流传感器", Min_Value := "Modbus_Data".电流传感器参数[0], Max_Value := "Modbus_Data".电流传感器参数[1], Project_amount => "Modbus_Data_Rapid".传感器标定值[7])
   END_RUNG
   // the same network as SCL:
   "Analog To Project amount"(Analog := "电流传感器",
                           Min_Value := "Modbus_Data".电流传感器参数[0],
                           Max_Value := "Modbus_Data".电流传感器参数[1],
                           Project_amount => "Modbus_Data_Rapid".传感器标定值[7]);
END_REGION
END_ORGANIZATION_BLOCK